FUNCTION_BLOCK RP_MOTOR (* Simple FB with one algorithm *)
  (* Standard: 61499-1 *)
  (* Version 1.0, 2025-07-17, vadim *)
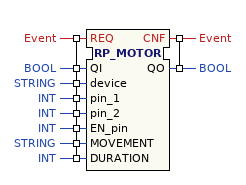
  EVENT_INPUT
    REQ WITH QI, pin_1, pin_2, EN_pin, DURATION, MOVEMENT, device; (* Normal Execution Request *)
  END_EVENT
  EVENT_OUTPUT
    CNF WITH QO; (* Execution Confirmation *)
  END_EVENT
  VAR_INPUT
    QI : BOOL; (* enable for cur. block *)
    device : STRING; (* device name *)
    pin_1 : INT; (* pin 1 *)
    pin_2 : INT; (* pin 2 *)
    EN_pin : INT; (* Enable pin *)
    MOVEMENT : STRING; (* forward/backward *)
    DURATION : INT; (* duration (ms) *)
  END_VAR
  VAR_OUTPUT
    QO : BOOL; (* Enable for next block *)
  END_VAR
  EC_STATES
    REQ : REQ -> CNF;
  END_STATES
  ALGORITHM REQ IN ST:

  END_ALGORITHM
END_FUNCTION_BLOCK
